	    REGION Niveaumessung
	        // Füllstand Versorgung Frischsäure
	        "Analogwert"(Deaktiviert:=FALSE,
	                                                                                                                                                                                                                                                                                                                                                                                                                                                                                                                                                                                                                                                                                                                                                                                                                                                                                                                                                                                                                                                                                                                                                                                                                                                                                                                                                                                                                                                                                                                                                                                                                                                                                                                                                                                                                                                                                                                                                                                                                                                                                                                                                                                                                                                                                                                                                                                                                                                                                                                                                                                                                                                                                                                                                                                                                                                                                                                                                                                                                                                                                                                                                                                                                                                                                                                                                                                                                                                                                                                                                                                                                                                                                                                                                                                                                                                                                                                                                                                                                                                                                                                                                                                                                                                                                                                                                                                                                                                                                                                                                                                                                                                                                                                                                                                                                                                                                                                                                                                                                                                                                                                                                                                                                                                                                                                                                                                                                                                                                                                                                                                                                                                                                                                                                                                                                                                                                                                                                                                                                                                                                                                                                                                                                                                                                                                                                                                                                                                                                                                                                                                                                                                                                                                                                                                                                                                                                                                                                                                                                                                                                                                                                                                                                                                                                                                                                                                                                                                                                                                                                                                                                                                                                                                                                                                                                                                                                                                                                                                                                                                                                                                                                                                                                                                                                                                                                                                                                                                                                                                                                                                                                                                                                                                                                                                                                                                                                                                                                                                                                                                                                                                                                                                                                                                                                                                                                                                                                                                                                                                                                                                                                                                                                                                                                                                                                                                                                                                                                                                                                                                                                                                                                                                                                                                                                                                                                                                                                                                                                                                                                                                                                                                                                                                                                                                                                                                                                                                                                                                                                                                                                                                                                                                                                                                                                                                                                                                                                                                                                                                                                                                                                                                                                                                                                                                                                                                                                                                                                                                                                                                                                                                                                                                                                                                                                                                                                                                                                                                                                                                                                                                                                                                                                                                                                                                                                                                                                                                                                                                                                                                                                                                                                                                                                                                                                                                                                                                                                                                                                                                                                                                                                                                                                                                                                                                                                                                                                                                                                                                                                                                                                                                                                                                                                                                                                                                                                                                                                                                                                                                                                                                                                                                                                                                                                                                                                                                                                                                                                                                                                                                                                                                                                                                                                                                                                                                                                                                                                                                                                                                                                                                                                                                                                                                                                                                                                                                                                                                                                                                                                                                                                                                                                                                                                                                                                                                                                                                                                                                                                                                                                                                                                                                                                                                                                                                                                                                                                                                                                                                                                                                                                                                                                                                                                                                                                                                                                                                                                                                                                                                                                                                                                                                                                                                                                                                                                                                                                                                                                                                                                                                                                                                                                                                                                                                                                                                                                                                                                                                                                                                                                                                                                                                                                                                                                                                                                                                                                                                                                                                                                                                                                                                                                                                                                                                                                                                                                                                                                                                                                                                                                                                                                                                                                                                                                                                                                                                                                                                                                                                                                                                                                                                                                                                                                                                                                                                                                                                                                                                                                                                                                                                                                                                                                                                                                                                                                                                                                                                                                                                                                                                                                                                                                                                                                                                                                                                                                                                                                                                                                                                                                                                                                                                                                                                                                                                                                                                                                                                                                                                                                                                                                                                                                                                                                                                                                                                                                                                                                                                                                                                                                                                                                                                                                                                                                                                                                                                                                                                                                                                                                                                                                                                                                                                                                                                                                                                                                                                                                                                                                                                                                                                                                                                                                                                                                                                                                                                                                                                                                                                                                                                                                                                                                                                                                                                                                                                                                                                                                                                                                                                                                                                                                                                                                                                                                                                                                                                                                                                                                                                                                                                                                                                                                                                                                                                                                                                                                                                                                                                                                                                                                                                                                                                                                                                                                                                                                                                                                                                                                                                                                                                                                                                                                                                                                                                                                                                                                                                                                                                                                                                                                                                                                                                                                                                                                                                                                                                                                                                                                                                                                                                                                                                                                                                                                                                                                                                                                                                                                                                                                                                                                                                                                                                                                                                                                                                                                                                                                                                                                                                                                                                                                                                                                                                                                                                                                                                                                                                                                                                                                                                                                                                                                                                                                                                                                                                                                                                                                                                                                                                                                                                                                                                                                                                                                                                                                                                                                                                                                                                                                                                                                                                                                                                                                                                                                                                                                                                                                                                                                                                                                                                                                                                                                                                                                                                                                                                                                                                                                                                                                                                                                                                                                                                                                                                                                                                                                                                                                                                                                                                                                                                                                                                                                                                                                                                                                                                                                                                                                                                                                                                                                                                                                                                                                                                                                                                                                                                                                                                                                                                                                                                                                                                                                                                                                                                                                                                                                                                                                                                                                                                                                                                                                                                                                                                                                                                                                                                                                                                                                                                                                                                                                                                                                                                                                                                                                                                                                                                                                                                                                                                                                                                                                                                                                                                                                                                                                                                                                                                                                                                                                                                                                                                                                                                                                                                                                                                                                                                                                                                                                                                                                                                                                                                                                                                                                                                                                                                                                                                                                                                                                                                                                                                                                                                                                                                                                                                                                                                                                                                                                                                                                                                                                                                                                                                                                                                                                                                                                                                                                                                                                                                                                                                                                                                                                                                                                                                                                                                                                                                                                                                                                                                                                                                                                                                                                                                                                                                                                                                                                                                                                                                                                                                                                                                                                                                                                                                                                                                                                                                                                                                                                                                                                                                                                                                                                                                                                                                                                                                                                                                                                                                                                                                                                                                                                                                                                                                                                                                                                                                                                                                                                                                                                                                                                                                                                                                                                                                                                                                                                                                                                                                                                                                                                                                                                                                                                                                                                                                                                                                                                                                                                                                                                                                                                                                                                                                                                                                                                                                                                                                                                                                                                                                                                                                                                                                                                                                                                                                                                                                                                                                                                                                                                                                                                                                                                                                                                                                                                                                                                                                                                                                                                                                                                                                                                                                                                                                                                                                                                                                                                                                                                                                                                                                                                                                                                                                                                                                                                                                                                                                                                                                                                                                                                                                                                                                                                                                                                                                                                                                                                                                                                                                                                                                                                                                                                                                                                                                                                                                                                                                                                                                                                                                                                                                                                                                                                                                                                                                                                                                                                                                                                                                                                                                                                                                                                                                                                                                                                                                                                                                                                                                                                                                                                                                                                                                                                                                                                                                                                                                                                                                                                                                                                                                                                                                                                                                                                                                                                                                                                                                                                                                                                                                                                                                                                                                                                                                                                                                                                                                                                                                                                                                                                                                                                                                                                                                                                                                                                                                                                                                                                                                                                                                                                                                                                                                                                                                                                                                                                                                                                                                                                                                                                                                                                                                                                                                                                                                                                                                                                                                                                                                                                                                                                                                                                                                                                                                                                                                                                                                                                                                                                                                                                                                                                                                                                                                                                                                                                                                                                                                                                                                                                                                                                                                                                                                                                                                                                                                                                                                                                                                                                                                                                                                                                                                                                                                                                                                                                                                                                                                                                                                                                                                                                                                                                                                                                                                                                                                                                                                                                                                                                                                                                                                                                                                                                                                                                                                                                                                                                                                                                                                                                                                                                                                                                                                                                                                                                                                                                                                                                                                                                                                                                                                                                                                                                                                                                                                                                                                                                                                                                                                                                                                                                                                                                                                                                                                                                                                                                                                                                                                                                                                                                                                                                                                                                                                                                                                                                                                                                                                                                                                                                                                                                                                                                                                                                                                                                                                                                                                                                                                                                                                                                                                                                                                                                                                                                                                                                                                                                                                                                                                                                                                                                                                                                                                                                                                                                                                                                                                                                                                                                                                                                                                                                                                                                                                                                                                                                                                                                                                                                                                                                                                                                                                                                                                                                                                                                                                                                                                                                                                                                                                                                                                                                                                                                                                                                                                                                                                                                                                                                                                                                                                                                                                                                                                                                                                                                                                                                                                                                                                                                                                                                                                                                                                                                                                                                                                                                                                                                                                                                                                                                                                                                                                                                                                                                                                                                                                                                                                                                                                                                                                                                                                                                                                                                                                                                                                                                                                                                                                                                                                                                                                                                                                                                                                                                                                                                                                                                                                                                                                                                                                                                                                                                                                                                                                                                                                                                                                                                                                                                                                                                                                                                                                                                                                                                                                                                                                                                                                                                                                                                                                                                                                                                                                                                                                                                                                                                                                                                                                                                                                                                                                                                                                                                                                                                                                                                                                                                                                                                                                                                                                                                                                                                                                                                                                                                                                                                                                                                                                                                                                                                                                                                                                                                                                                                                                                                                                                                                                                                                                                                                                                                                                                                                                                                                                                                                                                                                                                                                                                                                                                                                                                                                                                                                                                                                                                                                                                                                                                                                                                                                                                                                                                                                                                                                                                                                                                                                                                                                                                                                                                                                                                                                                                                                                                                                                                                                                                                                                                                                                                                                                                                                                                                                                                                                                                                                                                                                                                                                                                                                                                                                                                                                                                                                                                                                                                                                                                                                                                                                                                                                                                                                                                                                                                                                                                                                                                                                                                                                                                                                                                                                                                                                                                                                                                                                                                                                                                                                                                                                                                                                                                                                                                                                                                                                                                                                                                                                                                                                                                                                                                                                                                                                                                                                                                                                                                                                                                                                                                                                                                                                                                                                                                                                                                                                                                                                                                                                                                                                                                                                                                                                                                                                                                                                                                                                                                                                                                                                                                                                                                                                                                                                                                                                                                                                                                                                                                                                                                                                                                                                                                                                                                                                                                                                                                                                                                                                                                                                                                                                                                                                                                                                                                                                                                                                                                                                                                                                                                                                                                                                                                                      EW := "EW_Niv_GP01.BL30",
	                     Messbereich_Min := "Analogwerte"."Niv_GP01.BL30".MB_min,
	                     Messbereich_Max := "Analogwerte"."Niv_GP01.BL30".MB_max,
	                     UG_Alarm := "Analogwerte"."Niv_GP01.BL30".UG_Alarm,
	                     OG_Alarm := "Analogwerte"."Niv_GP01.BL30".OG_Alarm,
	                     GF := "Analogwerte"."Niv_GP01.BL30".GF,
	                     Al_Drahtbruch => "Analogwerte"."Niv_GP01.BL30".Drahtbruch,
	                     Al_MW_ausserhalb => "Analogwerte"."Niv_GP01.BL30".ungueltig,
	                     Messwert := "Panel".IW."Niv_GP01.BL30");
	        // Füllstand Entsorgung Altsäure
	        "Analogwert"(Deaktiviert:=FALSE,
	                        EW := "EW_Niv_GP02.BL31",
	                     Messbereich_Min := "Analogwerte"."Niv_GP02.BL31".MB_min,
	                     Messbereich_Max := "Analogwerte"."Niv_GP02.BL31".MB_max,
	                     UG_Alarm := "Analogwerte"."Niv_GP02.BL31".UG_Alarm,
	                     OG_Alarm := "Analogwerte"."Niv_GP02.BL31".OG_Alarm,
	                     GF := "Analogwerte"."Niv_GP02.BL31".GF,
	                     Al_Drahtbruch => "Analogwerte"."Niv_GP02.BL31".Drahtbruch,
	                     Al_MW_ausserhalb => "Analogwerte"."Niv_GP02.BL31".ungueltig,
	                     Messwert := "Panel".IW."Niv_GP02.BL31");
	     END_REGION
	// pH-Messung
	     "Analogwert"(Deaktiviert:=FALSE,
	             EW := "EW_LW_BE",
	             Messbereich_Min := "Analogwerte".pH_WR01.MB_min,
	             Messbereich_Max := "Analogwerte".pH_WR01.MB_max,
	             UG_Alarm := "Analogwerte".pH_WR01.UG_Alarm,
	             OG_Alarm := "Analogwerte".pH_WR01.OG_Alarm,
	             GF := "Analogwerte".pH_WR01.GF,
	             Al_Drahtbruch => "Analogwerte".pH_WR01.Drahtbruch,
	             Al_MW_ausserhalb => "Analogwerte".pH_WR01.ungueltig,
	             Messwert := "Panel".IW."pH_BE");
	END_IF;

	REGION Manipulator
	    IF "Imp_10Hz" THEN // 8x Wägezelle, 2x Last
	        "Analogwert"(Deaktiviert:=FALSE,
	                     EW := "EW_WZ_links_1",
	                     Messbereich_Min := "Analogwerte".WZ_1_1.MB_min,
	                     Messbereich_Max := "Analogwerte".WZ_1_1.MB_max,
	                     UG_Alarm := "Analogwerte".WZ_1_1.UG_Alarm,
	                     OG_Alarm := "Analogwerte".WZ_1_1.OG_Alarm,
	                     GF := "Analogwerte".WZ_1_1.GF,
	                     Al_Drahtbruch => "Analogwerte".WZ_1_1.Drahtbruch,
	                     Al_MW_ausserhalb => "Analogwerte".WZ_1_1.ungueltig,
	                     Messwert := "DI_FW_1".HELP.WZ_links_1);

	        "Analogwert"(Deaktiviert:=FALSE,
	                     EW := "EW_WZ_links_2",
	                     Messbereich_Min := "Analogwerte".WZ_1_2.MB_min,
	                     Messbereich_Max := "Analogwerte".WZ_1_2.MB_max,
	                     UG_Alarm := "Analogwerte".WZ_1_2.UG_Alarm,
	                     OG_Alarm := "Analogwerte".WZ_1_2.OG_Alarm,
	                     GF := "Analogwerte".WZ_1_2.GF,
	                     Al_Drahtbruch => "Analogwerte".WZ_1_2.Drahtbruch,
	                     Al_MW_ausserhalb => "Analogwerte".WZ_1_2.ungueltig,
	                     Messwert := "DI_FW_1".HELP.WZ_links_2);

	        "Analogwert"(Deaktiviert:=FALSE,
	                     EW := "EW_WZ_links_3",
	                     Messbereich_Min := "Analogwerte".WZ_1_3.MB_min,
	                     Messbereich_Max := "Analogwerte".WZ_1_3.MB_max,
	                     UG_Alarm := "Analogwerte".WZ_1_3.UG_Alarm,
	                     OG_Alarm := "Analogwerte".WZ_1_3.OG_Alarm,
	                     GF := "Analogwerte".WZ_1_3.GF,
	                     Al_Drahtbruch => "Analogwerte".WZ_1_3.Drahtbruch,
	                     Al_MW_ausserhalb => "Analogwerte".WZ_1_3.ungueltig,
	                     Messwert := "DI_FW_1".HELP.WZ_links_3);

	        "Analogwert"(Deaktiviert:=FALSE,
	                    EW := "EW_WZ_links_4",
	                     Messbereich_Min := "Analogwerte".WZ_1_4.MB_min,
	                     Messbereich_Max := "Analogwerte".WZ_1_4.MB_max,
	                     UG_Alarm := "Analogwerte".WZ_1_4.UG_Alarm,
	                     OG_Alarm := "Analogwerte".WZ_1_4.OG_Alarm,
	                     GF := "Analogwerte".WZ_1_4.GF,
	                     Al_Drahtbruch => "Analogwerte".WZ_1_4.Drahtbruch,
	                     Al_MW_ausserhalb => "Analogwerte".WZ_1_4.ungueltig,
	                     Messwert := "DI_FW_1".HELP.WZ_links_4);

	        "Analogwert"(Deaktiviert:=FALSE,
	                     EW := "EW_WZ_rechts_1",
	                     Messbereich_Min := "Analogwerte".WZ_2_1.MB_min,
	                     Messbereich_Max := "Analogwerte".WZ_2_1.MB_max,
	                     UG_Alarm := "Analogwerte".WZ_2_1.UG_Alarm,
	                     OG_Alarm := "Analogwerte".WZ_2_1.OG_Alarm,
	                     GF := "Analogwerte".WZ_2_1.GF,
	                     Al_Drahtbruch => "Analogwerte".WZ_2_1.Drahtbruch,
	                     Al_MW_ausserhalb => "Analogwerte".WZ_2_1.ungueltig,
	                     Messwert := "DI_FW_1".HELP.WZ_rechts_1);

	        "Analogwert"(Deaktiviert := FALSE,
	                     EW := "EW_WZ_rechts_2",
	                     Messbereich_Min := "Analogwerte".WZ_2_2.MB_min,
	                     Messbereich_Max := "Analogwerte".WZ_2_2.MB_max,
	                     UG_Alarm := "Analogwerte".WZ_2_2.UG_Alarm,
	                     OG_Alarm := "Analogwerte".WZ_2_2.OG_Alarm,
	                     GF := "Analogwerte".WZ_2_2.GF,
	                     Al_Drahtbruch => "Analogwerte".WZ_2_2.Drahtbruch,
	                     Al_MW_ausserhalb => "Analogwerte".WZ_2_2.ungueltig,
	                     Messwert := "DI_FW_1".HELP.WZ_rechts_2);

	        "Analogwert"(Deaktiviert := FALSE,
	                     EW := "EW_WZ_rechts_3",
	                     Messbereich_Min := "Analogwerte".WZ_2_3.MB_min,
	                     Messbereich_Max := "Analogwerte".WZ_2_3.MB_max,
	                     UG_Alarm := "Analogwerte".WZ_2_3.UG_Alarm,
	                     OG_Alarm := "Analogwerte".WZ_2_3.OG_Alarm,
	                     GF := "Analogwerte".WZ_2_3.GF,
	                     Al_Drahtbruch => "Analogwerte".WZ_2_3.Drahtbruch,
	                     Al_MW_ausserhalb => "Analogwerte".WZ_2_3.ungueltig,
	                     Messwert := "DI_FW_1".HELP.WZ_rechts_3);

	        "Analogwert"(Deaktiviert := FALSE,
	                     EW := "EW_WZ_rechts_4",
	                     Messbereich_Min := "Analogwerte".WZ_2_4.MB_min,
	                     Messbereich_Max := "Analogwerte".WZ_2_4.MB_max,
	                     UG_Alarm := "Analogwerte".WZ_2_4.UG_Alarm,
	                     OG_Alarm := "Analogwerte".WZ_2_4.OG_Alarm,
	                     GF := "Analogwerte".WZ_2_4.GF,
	                     Al_Drahtbruch => "Analogwerte".WZ_2_4.Drahtbruch,
	                     Al_MW_ausserhalb => "Analogwerte".WZ_2_4.ungueltig,
	                     Messwert := "DI_FW_1".HELP.WZ_rechts_4);

	        "Analogwert"(Deaktiviert := FALSE,
	                     EW := "EW_Last_links",
	                     Messbereich_Min := "Analogwerte".Last_1.MB_min,
	                     Messbereich_Max := "Analogwerte".Last_1.MB_max,
	                     UG_Alarm := "Analogwerte".Last_1.UG_Alarm,
	                     OG_Alarm := "Analogwerte".Last_1.OG_Alarm,
	                     GF := "Analogwerte".Last_1.GF,
	                     Al_Drahtbruch => "Analogwerte".Last_1.Drahtbruch,
	                     Al_MW_ausserhalb => "Analogwerte".Last_1.ungueltig,
	                     Messwert := "DI_FW_1".HELP.Last_1);

	        "Analogwert"(Deaktiviert:=FALSE,
	                     EW := "EW_Last_rechts",
	                     Messbereich_Min := "Analogwerte".Last_2.MB_min,
	                     Messbereich_Max := "Analogwerte".Last_2.MB_max,
	                     UG_Alarm := "Analogwerte".Last_2.UG_Alarm,
	                     OG_Alarm := "Analogwerte".Last_2.OG_Alarm,
	                     GF := "Analogwerte".Last_2.GF,
	                     Al_Drahtbruch => "Analogwerte".Last_2.Drahtbruch,
	                     Al_MW_ausserhalb => "Analogwerte".Last_2.ungueltig,
	                     Messwert := "DI_FW_1".HELP.Last_2);
	    END_IF;

	END_REGION

END_FUNCTION

